// TIA Portal project "2020-10-02_LuceConSensori" (V16)

(* hardware
DEVICE "S7-1200 station_1"  S7-1200 Station
   slot 0: "Telaio di montaggio_0"  S7-1200 Rack  Rack  V1.0
   slot 1: "PLC_1"  CPU 1215C DC/DC/DC  6ES7 215-1AG40-0XB0  V4.4
*)

// ===== PLC "PLC_1"  CPU 1215C DC/DC/DC =====

VAR_GLOBAL   // PLC tag table "Tabella delle variabili standard"
   "s1" AT %I0.0 : Bool;
   "s2" AT %I0.1 : Bool;
   "s3" AT %I0.2 : Bool;
   "luce" AT %Q0.0 : Bool;
END_VAR

ORGANIZATION_BLOCK "Main"   // OB1, LAD, ProgramCycle
TITLE = "Main Program Sweep (Cycle)"
{ S7_Optimized_Access := 'TRUE' }
VERSION : 0.1
   VAR_INPUT
      Initial_Call : Bool;   // Initial call of this OB
      Remanence : Bool;   // =True, if remanent data are available
   END_VAR
BEGIN

REGION Network 1
   // setto(accendo) la luce quando la maggioranza dei sensori mi da 0(buio)
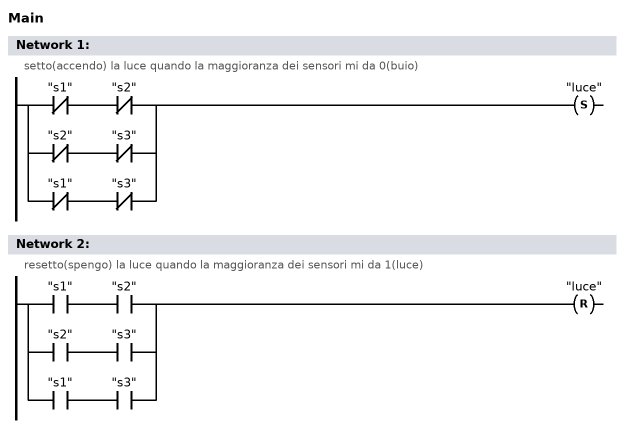
   RUNG wire#powerrail
      I_Contact( "s1" )
      I_Contact( "s2" )
      wire#w1
      S_Coil( "luce" )
   END_RUNG
   RUNG wire#powerrail
      I_Contact( "s2" )
      I_Contact( "s3" )
   END_RUNG wire#w1
   RUNG wire#powerrail
      I_Contact( "s1" )
      I_Contact( "s3" )
   END_RUNG wire#w1
   // the same network as SCL:
   IF (NOT "s1" AND NOT "s2") OR (NOT "s2" AND NOT "s3") OR (NOT "s1" AND NOT "s3") THEN
       "luce" := TRUE;
   END_IF;
END_REGION

REGION Network 2
   // resetto(spengo) la luce quando la maggioranza dei sensori mi da 1(luce)
   RUNG wire#powerrail
      Contact( "s1" )
      Contact( "s2" )
      wire#w1
      R_Coil( "luce" )
   END_RUNG
   RUNG wire#powerrail
      Contact( "s2" )
      Contact( "s3" )
   END_RUNG wire#w1
   RUNG wire#powerrail
      Contact( "s1" )
      Contact( "s3" )
   END_RUNG wire#w1
   // the same network as SCL:
   IF ("s1" AND "s2") OR ("s2" AND "s3") OR ("s1" AND "s3") THEN "luce" := FALSE; END_IF;
END_REGION
END_ORGANIZATION_BLOCK